// TIA Portal V20 export
DATA_BLOCK "DB_DigitalOutputs"   // DB2103
// stored: AutoNumber false, InstanceOfName FB_DigitalOutputs, InstanceOfType FB
"FB_DigitalOutputs"
   // VAR
   //    sFreeQ0_0 : "FB_DigitalOutput";
   //    sOperatingCounter : "FB_DigitalOutput";
   //    sGeneralAirValve : "FB_DigitalOutput";
   //    sSmartLineDisable : "FB_DigitalOutput";
   //    sMachineLight : "FB_DigitalOutput";
   //    sMachineLightBack : "FB_DigitalOutput";
   //    sLightTowerOrange : "FB_DigitalOutput";
   //    sLightTowerRed : "FB_DigitalOutput";
   //    sLightTowerBlue : "FB_DigitalOutput";
   //    sLightTowerGreen : "FB_DigitalOutput";
   //    sLightTowerWhite : "FB_DigitalOutput";
   //    sBacklight : "FB_DigitalOutput";
   //    sFreeQ1_4 : "FB_DigitalOutput";
   //    sInfeedON : "FB_DigitalOutput";
   //    sAxisActivation : "FB_DigitalOutput";
   //    sBuzzerActivation : "FB_DigitalOutput";
   //    sElbaronPowerON : "FB_DigitalOutput";
   //    sObservationCameraLight : "FB_DigitalOutput";
   //    sLaserExternalDoorOpening : "FB_DigitalOutput";
   //    sCoolingStart : "FB_DigitalOutput";
   //    sX_AxisBrakeActivation : "FB_DigitalOutput";
   //    sY_AxisBrakeActivation : "FB_DigitalOutput";
   //    sAxisB_TeachInClampingPart : "FB_DigitalOutput";
   //    sEPO_UPS : "FB_DigitalOutput";
   //    sHeadLaserStart : "FB_DigitalOutput";
   //    sHeadLaserStop : "FB_DigitalOutput";
   //    sAxis2_PowerContactor : "FB_DigitalOutput";
   //    sGasAssistOn : "FB_DigitalOutput";
   //    sSmartLineReset : "FB_DigitalOutput";
   //    sXY_AxisPowerContactor : "FB_DigitalOutput";
   //    sLaserAirPressureProcess : "FB_DigitalOutput";
   //    sBus60V_PowerContactor : "FB_DigitalOutput";
   //    sFreeQ4_0 : "FB_DigitalOutput";
   //    sFreeQ4_1 : "FB_DigitalOutput";
   //    sFreeQ4_2 : "FB_DigitalOutput";
   //    sFreeQ4_3 : "FB_DigitalOutput";
   //    sLoadClampClosing : "FB_DigitalOutput";
   //    sLoadClampOpening : "FB_DigitalOutput";
   //    sUnloadClampClosing : "FB_DigitalOutput";
   //    sUnloadClampOpening : "FB_DigitalOutput";
   //    sClampingOpening : "FB_DigitalOutput";
   //    sClampingClosing : "FB_DigitalOutput";
   //    sB_AxisBrakeRelease : "FB_DigitalOutput";
   //    sSuction : "FB_DigitalOutput";
   //    sFreeQ5_4 : "FB_DigitalOutput";
   //    sFreeQ5_5 : "FB_DigitalOutput";
   //    sFreeQ5_6 : "FB_DigitalOutput";
   //    sFreeQ5_7 : "FB_DigitalOutput";
   //    sExternalGateClosing : "FB_DigitalOutput";
   //    sExternalGateOpening : "FB_DigitalOutput";
   //    sInternalGateClosing : "FB_DigitalOutput";
   //    sInternalGateOpening : "FB_DigitalOutput";
   //    sPowerMeterRetract : "FB_DigitalOutput";
   //    sPowerMeterAdvance : "FB_DigitalOutput";
   //    sBlowing : "FB_DigitalOutput";
   //    sFreeQ8_7 : "FB_DigitalOutput";
   //    sFreeQ9_0 : "FB_DigitalOutput";
   //    sFreeQ9_1 : "FB_DigitalOutput";
   //    sFreeQ9_2 : "FB_DigitalOutput";
   //    sFreeQ9_3 : "FB_DigitalOutput";
   //    sFreeQ9_4 : "FB_DigitalOutput";
   //    sFreeQ9_5 : "FB_DigitalOutput";
   //    sFreeQ9_6 : "FB_DigitalOutput";
   //    sFreeQ9_7 : "FB_DigitalOutput";
   //    sSonplasDiagDPCoupler { S7_SetPoint := 'True'} : "FB_DigitalOutput";
   //    sSonplasReady { S7_SetPoint := 'True'} : "FB_DigitalOutput";
   //    sSonplasNoEStop { S7_SetPoint := 'True'} : "FB_DigitalOutput";
   //    sSonplasDoorsClosed { S7_SetPoint := 'True'} : "FB_DigitalOutput";
   //    sSonplasRunError { S7_SetPoint := 'True'} : "FB_DigitalOutput";
   //    sSonplasFreeQ200_5 { S7_SetPoint := 'True'} : "FB_DigitalOutput";
   //    sSonplasFreeQ200_6 { S7_SetPoint := 'True'} : "FB_DigitalOutput";
   //    sSonplasFreeQ200_7 { S7_SetPoint := 'True'} : "FB_DigitalOutput";
   //    sSonplasFreeQ201_0 { S7_SetPoint := 'True'} : "FB_DigitalOutput";
   //    sSonplasFreeQ201_1 { S7_SetPoint := 'True'} : "FB_DigitalOutput";
   //    sSonplasFreeQ201_2 { S7_SetPoint := 'True'} : "FB_DigitalOutput";
   //    sSonplasFreeQ201_3 { S7_SetPoint := 'True'} : "FB_DigitalOutput";
   //    sSonplasFreeQ201_4 { S7_SetPoint := 'True'} : "FB_DigitalOutput";
   //    sSonplasFreeQ201_5 { S7_SetPoint := 'True'} : "FB_DigitalOutput";
   //    sSonplasFreeQ201_6 { S7_SetPoint := 'True'} : "FB_DigitalOutput";
   //    sSonplasFreeQ201_7 { S7_SetPoint := 'True'} : "FB_DigitalOutput";
   //    sSonplasShuttle1InPos { S7_SetPoint := 'True'} : "FB_DigitalOutput";
   //    sSonplasFreeQ202_1 { S7_SetPoint := 'True'} : "FB_DigitalOutput";
   //    sSonplasFreeQ202_2 { S7_SetPoint := 'True'} : "FB_DigitalOutput";
   //    sSonplasFreeQ202_3 { S7_SetPoint := 'True'} : "FB_DigitalOutput";
   //    sSonplasFreeQ202_4 { S7_SetPoint := 'True'} : "FB_DigitalOutput";
   //    sSonplasFreeQ202_5 { S7_SetPoint := 'True'} : "FB_DigitalOutput";
   //    sSonplasPart1OK { S7_SetPoint := 'True'} : "FB_DigitalOutput";
   //    sSonplasPart1NOK { S7_SetPoint := 'True'} : "FB_DigitalOutput";
   //    sSonplasShuttle2InPos { S7_SetPoint := 'True'} : "FB_DigitalOutput";
   //    sSonplasFreeQ203_1 { S7_SetPoint := 'True'} : "FB_DigitalOutput";
   //    sSonplasFreeQ203_2 { S7_SetPoint := 'True'} : "FB_DigitalOutput";
   //    sSonplasFreeQ203_3 { S7_SetPoint := 'True'} : "FB_DigitalOutput";
   //    sSonplasFreeQ203_4 { S7_SetPoint := 'True'} : "FB_DigitalOutput";
   //    sSonplasFreeQ203_5 { S7_SetPoint := 'True'} : "FB_DigitalOutput";
   //    sSonplasPart2OK { S7_SetPoint := 'True'} : "FB_DigitalOutput";
   //    sSonplasPart2NOK { S7_SetPoint := 'True'} : "FB_DigitalOutput";
   //    sSonplasResultAccepted { S7_SetPoint := 'True'} : "FB_DigitalOutput";
   //    sSonplasFreeQ244_1 { S7_SetPoint := 'True'} : "FB_DigitalOutput";
   //    sSonplasFreeQ244_2 { S7_SetPoint := 'True'} : "FB_DigitalOutput";
   //    sSonplasFreeQ244_3 { S7_SetPoint := 'True'} : "FB_DigitalOutput";
   //    sSonplasFreeQ244_4 { S7_SetPoint := 'True'} : "FB_DigitalOutput";
   //    sSonplasFreeQ244_5 { S7_SetPoint := 'True'} : "FB_DigitalOutput";
   //    sSonplasFreeQ244_6 { S7_SetPoint := 'True'} : "FB_DigitalOutput";
   //    sSonplasFreeQ244_7 { S7_SetPoint := 'True'} : "FB_DigitalOutput";
   // END_VAR
BEGIN
END_DATA_BLOCK
